Fanuc KAREL source: kd00024.KL

-- PROVISIONAL review KL for V770-1; original PC SHA256 175f379fb681c61fca166f6c6167564000903401805cb65dc46720a69dc220e8
-- Incomplete behavior may be omitted. Consult companion uncertainty JSON. Do not deploy.
PROGRAM KD00024
%NOLOCKGROUP
VAR
  I : INTEGER
  J : INTEGER
  B : BOOLEAN
  R : REAL
  S : STRING[80]
BEGIN
  -- UNRESOLVED_PC offsets 5-12; opcodes 9D,23
  -- UNRESOLVED_PC offsets 17-50; opcodes 9D,81,18,22,2E,21,54,12,22,9D,13,04
  -- UNRESOLVED_PC offsets 55-59; opcodes 7F
END KD00024
